// TIA Portal project "testeMaqEst" (V17)
// HARDWARE PADRAO CLP, INTERFACES E IHM

(* hardware
DEVICE "S7-1500/ET200MP station_1"  S7-1500 station
   slot 0: "Rail_0"  Rack  6ES7 590-1***0-0AA0
   slot 1: "PLC_1"  CPU 1516-3 PN/DP  6ES7 516-3AN01-0AB0  V2.9
      slot 3: "CPU display_1"  6ES7591-1BA00-0AA0
      slot 32768: "PROFINET interface_1"  X1
      slot 33024: "PROFINET interface_2"  X2
      slot 33280: "DP interface_1"  X3
      slot 34817: "Virtual CP interface port_1"  Virtual CP interface port  Virtual CP interface port
   slot 2: "DI 32x24VDC HF_1"  DI 32x24VDC HF  6ES7 521-1BL00-0AB0  V2.1
   slot 3: "DQ 32x24VDC/0.5A HF_1"  DQ 32x24VDC/0.5A HF  6ES7 522-1BL01-0AB0  V1.0
   slot 4: "AI 8xU/I/RTD/TC ST_1"  AI 8xU/I/RTD/TC ST  6ES7 531-7KF00-0AB0  V2.0
   slot 5: "AQ 4xU/I ST_1"  AQ 4xU/I ST  6ES7 532-5HD00-0AB0  V2.0
DEVICE "HMI_1"  KTP700 Basic PN
   slot 0: "HMI_1"  KTP700 Basic PN  6AV2 123-2GB03-0AX0  14.0.1.0
   slot 1: "HMI_RT_1"  KTP700 Basic PN  6AV2 123-2GB03-0AX0  14.0.1.0
   slot 5: "HMI_1.IE_CP_1"  PROFINET Interface  14.0.1.0
      slot 1: "PROFINET Interface_1"  PROFINET Interface
         slot 1: "Port_1"  Port
*)

// ===== PLC "PLC_1"  CPU 1516-3 PN/DP =====

VAR_GLOBAL   // PLC tag table "Default tag table"
   "Clock_Byte" AT %MB100 : Byte;
   "Clock_10Hz" AT %M100.0 : Bool;
   "Clock_5Hz" AT %M100.1 : Bool;
   "Clock_2.5Hz" AT %M100.2 : Bool;
   "Clock_2Hz" AT %M100.3 : Bool;
   "Clock_1.25Hz" AT %M100.4 : Bool;
   "Clock_1Hz" AT %M100.5 : Bool;
   "Clock_0.625Hz" AT %M100.6 : Bool;
   "Clock_0.5Hz" AT %M100.7 : Bool;
END_VAR

VAR_GLOBAL   // PLC tag table "ENTRADAS"
   "modo" AT %I0.1 : Bool;
   "on" AT %I0.2 : Bool;
   "RA" AT %I1.0 : Bool;
   "AA" AT %I1.1 : Bool;
   "RB" AT %I1.2 : Bool;
   "AB" AT %I1.3 : Bool;
END_VAR

VAR_GLOBAL   // PLC tag table "SAIDAS"
   "EVA" AT %Q0.0 : Bool;
   "EVB" AT %Q0.1 : Bool;
END_VAR

DATA_BLOCK "teste"   // DB1
{ S7_Optimized_Access := 'TRUE' }
VERSION : 0.1
   VAR
      estado : Int;
   END_VAR
BEGIN
END_DATA_BLOCK

// folder: System blocks/Program resources

DATA_BLOCK "tmr0"   // DB2
{ S7_Optimized_Access := 'TRUE' }
AUTHOR : Simatic
FAMILY : IEC
NAME : IEC_TMR
VERSION : 1.0
// stored: InstanceOfName IEC_TIMER
"IEC_TIMER"
BEGIN
END_DATA_BLOCK

// folder: (top level)

FUNCTION "A+B+B-A-" : Void   // FC1, LAD
{ S7_Optimized_Access := 'TRUE' }
VERSION : 0.1
   VAR_TEMP   // added for the SCL form of the ladder/FBD networks
      _w1 : Bool;
   END_VAR
BEGIN

REGION Network 1: T0
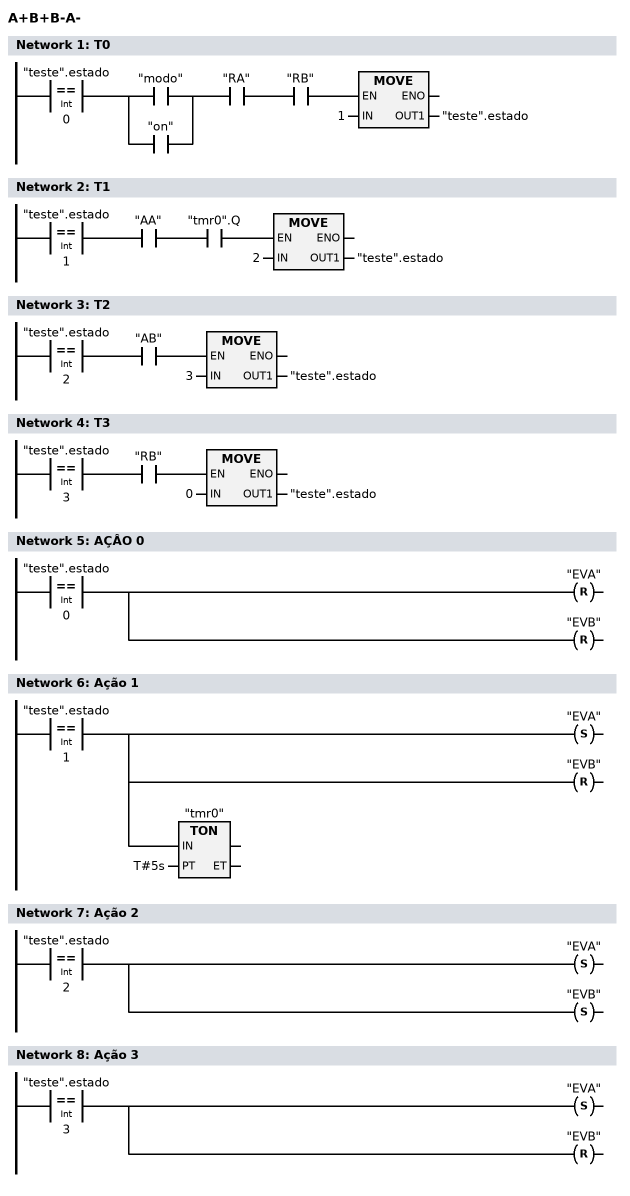
   RUNG wire#powerrail
      { S7_Templates := "SrcType := Int" } EQ_Contact(in1 := "teste".estado, in2 := 0)
      wire#w1
      Contact( "modo" )
      wire#w2
      Contact( "RA" )
      Contact( "RB" )
      Move(in := 1, out1 => "teste".estado)
   END_RUNG
   RUNG wire#w1
      Contact( "on" )
   END_RUNG wire#w2
   // the same network as SCL:
   IF ("teste".estado = 0) AND ("modo" OR "on") AND "RA" AND "RB" THEN "teste".estado := 1; END_IF;
END_REGION

REGION Network 2: T1
   RUNG wire#powerrail
      { S7_Templates := "SrcType := Int" } EQ_Contact(in1 := "teste".estado, in2 := 1)
      Contact( "AA" )
      Contact( "tmr0".Q )
      Move(in := 2, out1 => "teste".estado)
   END_RUNG
   // the same network as SCL:
   IF ("teste".estado = 1) AND "AA" AND "tmr0".Q THEN "teste".estado := 2; END_IF;
END_REGION

REGION Network 3: T2
   RUNG wire#powerrail
      { S7_Templates := "SrcType := Int" } EQ_Contact(in1 := "teste".estado, in2 := 2)
      Contact( "AB" )
      Move(in := 3, out1 => "teste".estado)
   END_RUNG
   // the same network as SCL:
   IF ("teste".estado = 2) AND "AB" THEN "teste".estado := 3; END_IF;
END_REGION

REGION Network 4: T3
   RUNG wire#powerrail
      { S7_Templates := "SrcType := Int" } EQ_Contact(in1 := "teste".estado, in2 := 3)
      Contact( "RB" )
      Move(in := 0, out1 => "teste".estado)
   END_RUNG
   // the same network as SCL:
   IF ("teste".estado = 3) AND "RB" THEN "teste".estado := 0; END_IF;
END_REGION

REGION Network 5: AÇÂO 0
   RUNG wire#powerrail
      { S7_Templates := "SrcType := Int" } EQ_Contact(in1 := "teste".estado, in2 := 0)
      wire#w1
      R_Coil( "EVA" )
   END_RUNG
   RUNG wire#w1
      R_Coil( "EVB" )
   END_RUNG
   // the same network as SCL:
   IF "teste".estado = 0 THEN
       "EVA" := FALSE;
       "EVB" := FALSE;
   END_IF;
END_REGION

REGION Network 6: Ação 1
   #_w1 := "teste".estado = 1;
   IF #_w1 THEN
       "EVA" := TRUE;
       "EVB" := FALSE;
   END_IF;
   "tmr0".TON(IN := #_w1, PT := T#5s);
END_REGION

REGION Network 7: Ação 2
   RUNG wire#powerrail
      { S7_Templates := "SrcType := Int" } EQ_Contact(in1 := "teste".estado, in2 := 2)
      wire#w1
      S_Coil( "EVA" )
   END_RUNG
   RUNG wire#w1
      S_Coil( "EVB" )
   END_RUNG
   // the same network as SCL:
   IF "teste".estado = 2 THEN
       "EVA" := TRUE;
       "EVB" := TRUE;
   END_IF;
END_REGION

REGION Network 8: Ação 3
   RUNG wire#powerrail
      { S7_Templates := "SrcType := Int" } EQ_Contact(in1 := "teste".estado, in2 := 3)
      wire#w1
      S_Coil( "EVA" )
   END_RUNG
   RUNG wire#w1
      R_Coil( "EVB" )
   END_RUNG
   // the same network as SCL:
   IF "teste".estado = 3 THEN
       "EVA" := TRUE;
       "EVB" := FALSE;
   END_IF;
END_REGION
END_FUNCTION

ORGANIZATION_BLOCK "Main"   // OB1, LAD, ProgramCycle
TITLE = "Main Program Sweep (Cycle)"
{ S7_Optimized_Access := 'TRUE' }
VERSION : 0.1
   VAR_INPUT
      Initial_Call : Bool;   // Initial call of this OB
      Remanence : Bool;   // =True, if remanent data are available
   END_VAR
BEGIN

REGION Network 1
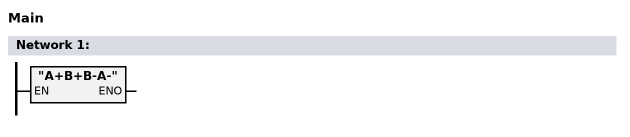
   RUNG wire#powerrail
      "A+B+B-A-"()
   END_RUNG
   // the same network as SCL:
   "A+B+B-A-"();
END_REGION
END_ORGANIZATION_BLOCK

(* ===== HMI "HMI_RT_1" =====
system functions are stored by id; their names below are inferred from use
connection "HMI_Connection_1": ETHERNET, SMART_S7_1500_OMS

Template "Template_1" 800x480
   Button "Exit" at 714,429 size 71x50; TextOff 'Exit'; PictureOff "ExitRuntime_KTP700_Basic_PN_TR"; PictureOn "ExitRuntime_KTP700_Basic_PN_TR"
      on Release: StopRuntime(0)
   Button "Template_Button" at 614,429 size 71x50; TextOff 'Text'
   Button "Template_Button_1" at 514,429 size 71x50; TextOff 'Text'
   Button "Template_Button_2" at 414,429 size 71x50; TextOff 'Text'
   Button "Template_Button_3" at 314,429 size 71x50; TextOff 'Text'
   Button "Template_Button_4" at 214,429 size 71x50; TextOff 'Text'
   Button "Template_Button_5" at 114,429 size 71x50; TextOff 'Text'
   Button "Start screen" at 14,429 size 71x50; TextOff 'Start screen'; PictureOff "NavigateHome_KTP700_Basic_PN_TR"; PictureOn "NavigateHome_KTP700_Basic_PN_TR"
      on Release: ActivateScreen("Root screen", 0)

screen "Root screen" 800x480, template "Template_1"
   TextField "HmiScreenItemData" at 80,200 size 640x25; Text 'PROJETO BASE ADS'
*)